// TIA Portal V20 export
DATA_BLOCK "GLOBAL_VALVE_HMI_IF_DB"   // DB220
{ S7_Optimized_Access := 'TRUE' }
// stored: AutoNumber false, MemoryReserve 100
   VAR RETAIN
      Valve { S7_SetPoint := 'True'} : Array[0..20] of "VALVE_HMI_UDT";
   END_VAR
BEGIN
   // Valve[1] : 左外上下缸
   // Valve[2] : 左外吸盘真空阀
END_DATA_BLOCK
